(* CODESYS project DigitalOutput_0.0.2.library
   Version: 0.0.2
   Title: DigitalOutput
   Author: Ali Alam
   Placeholder: DigitalOutput
   Company: Promise Robotics

Project tree, tasks and I/O mapping:
  libraries: Tc2_Standard, * (Beckhoff Automation GmbH); Tc2_System, * (Beckhoff Automation GmbH)
  DUTs/
  GVLs/
  POUs/
    function block FB_DigitalOutput [ST]: P_OperatorControl, P_OperatorValue, P_Output, SetOutput
    interface ITF_DigitalOutput: P_OperatorControl, P_OperatorValue, P_Output, SetOutput
  VISUs/
*)

// POUs/FB_DigitalOutput
FUNCTION_BLOCK FB_DigitalOutput IMPLEMENTS ITF_DigitalOutput
VAR
	{ attribute 'TcHmiSymbol.AddSymbol' }
	Output AT %Q*   	: BOOL;
	{ attribute 'TcHmiSymbol.AddSymbol' }
	OperatorControl 	: BOOL := FALSE;
	{ attribute 'TcHmiSymbol.AddSymbol' }
	OperatorValue		: BOOL; 
END_VAR

PROPERTY P_OperatorControl : BOOL
GET
P_OperatorControl := OperatorControl;
END_GET
SET
OperatorControl := P_OperatorControl;
END_SET
END_PROPERTY

PROPERTY P_OperatorValue : BOOL
GET
P_OperatorValue := OperatorValue;
END_GET
SET
OperatorValue := P_OperatorValue;
END_SET
END_PROPERTY

PROPERTY P_Output : BOOL
GET
P_Output := Output;
END_GET
END_PROPERTY

METHOD PUBLIC SetOutput : BOOL
VAR_INPUT
	Requested	: BOOL;
END_VAR
IF OperatorControl THEN
	Output := OperatorValue;
ELSE
	Output := Requested;
END_IF
END_METHOD

END_FUNCTION_BLOCK

// POUs/ITF_DigitalOutput
INTERFACE ITF_DigitalOutput

PROPERTY P_OperatorControl : BOOL
GET
END_GET
SET
END_SET
END_PROPERTY

PROPERTY P_OperatorValue : BOOL
GET
END_GET
SET
END_SET
END_PROPERTY

PROPERTY P_Output : BOOL
GET
END_GET
END_PROPERTY

METHOD SetOutput : BOOL
VAR_INPUT
	Requested	: BOOL;
END_VAR
END_METHOD

END_INTERFACE
